FUNCTION_BLOCK FB_PVFEEDIN_CALC (* Composite Function Block Type *)
  (* Standard: 61499-2 *)
  (* Version 0.0, 2017-06-15, Marc Jakobi, HTW Berlin *)
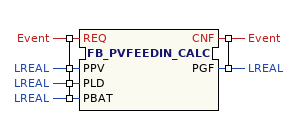
  EVENT_INPUT
    REQ WITH PPV, PLD, PBAT; (* Normal Execution Request *)
  END_EVENT
  EVENT_OUTPUT
    CNF WITH PGF; (* Execution Confirmation *)
  END_EVENT
  VAR_INPUT
    PPV : LREAL; (* PV power *)
    PLD : LREAL; (* Load *)
    PBAT : LREAL; (* Battery power (positive = charge, negative = discharge) *)
  END_VAR
  VAR_OUTPUT
    PGF : LREAL; (* Grid feed-in power *)
  END_VAR
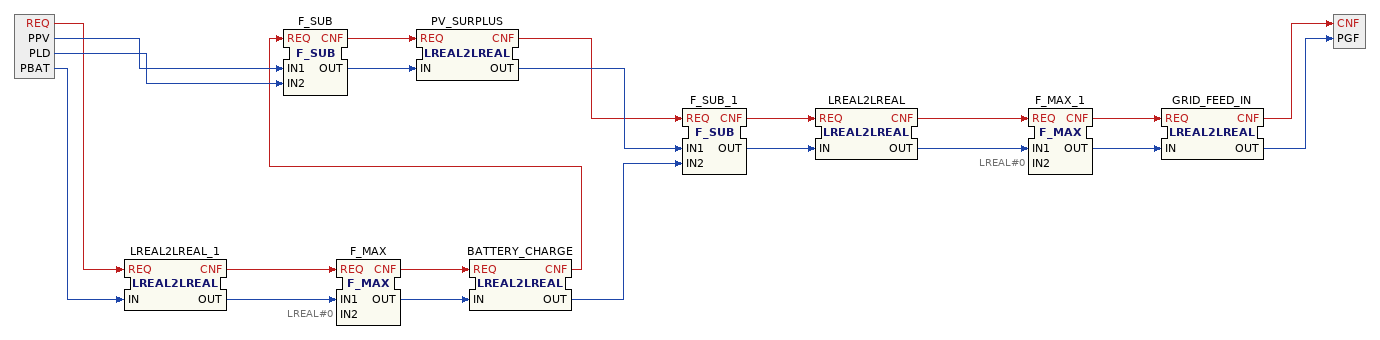
  FBS
    F_SUB : F_SUB;
    F_SUB_1 : F_SUB;
    PV_SURPLUS : LREAL2LREAL;
    F_MAX : F_MAX(IN2 := LREAL#0);
    LREAL2LREAL_1 : LREAL2LREAL;
    BATTERY_CHARGE : LREAL2LREAL;
    F_MAX_1 : F_MAX(IN2 := LREAL#0);
    LREAL2LREAL : LREAL2LREAL;
    GRID_FEED_IN : LREAL2LREAL;
  END_FBS
  EVENT_CONNECTIONS
    F_SUB.CNF TO PV_SURPLUS.REQ;
    PV_SURPLUS.CNF TO F_SUB_1.REQ;
    REQ TO LREAL2LREAL_1.REQ;
    LREAL2LREAL_1.CNF TO F_MAX.REQ;
    F_MAX.CNF TO BATTERY_CHARGE.REQ;
    BATTERY_CHARGE.CNF TO F_SUB.REQ;
    F_SUB_1.CNF TO LREAL2LREAL.REQ;
    LREAL2LREAL.CNF TO F_MAX_1.REQ;
    F_MAX_1.CNF TO GRID_FEED_IN.REQ;
    GRID_FEED_IN.CNF TO CNF;
  END_CONNECTIONS
  DATA_CONNECTIONS
    PPV TO F_SUB.IN1;
    PLD TO F_SUB.IN2;
    F_SUB.OUT TO PV_SURPLUS.IN;
    PV_SURPLUS.OUT TO F_SUB_1.IN1;
    PBAT TO LREAL2LREAL_1.IN;
    LREAL2LREAL_1.OUT TO F_MAX.IN1;
    F_MAX.OUT TO BATTERY_CHARGE.IN;
    BATTERY_CHARGE.OUT TO F_SUB_1.IN2;
    F_SUB_1.OUT TO LREAL2LREAL.IN;
    LREAL2LREAL.OUT TO F_MAX_1.IN1;
    F_MAX_1.OUT TO GRID_FEED_IN.IN;
    GRID_FEED_IN.OUT TO PGF;
  END_CONNECTIONS
END_FUNCTION_BLOCK
